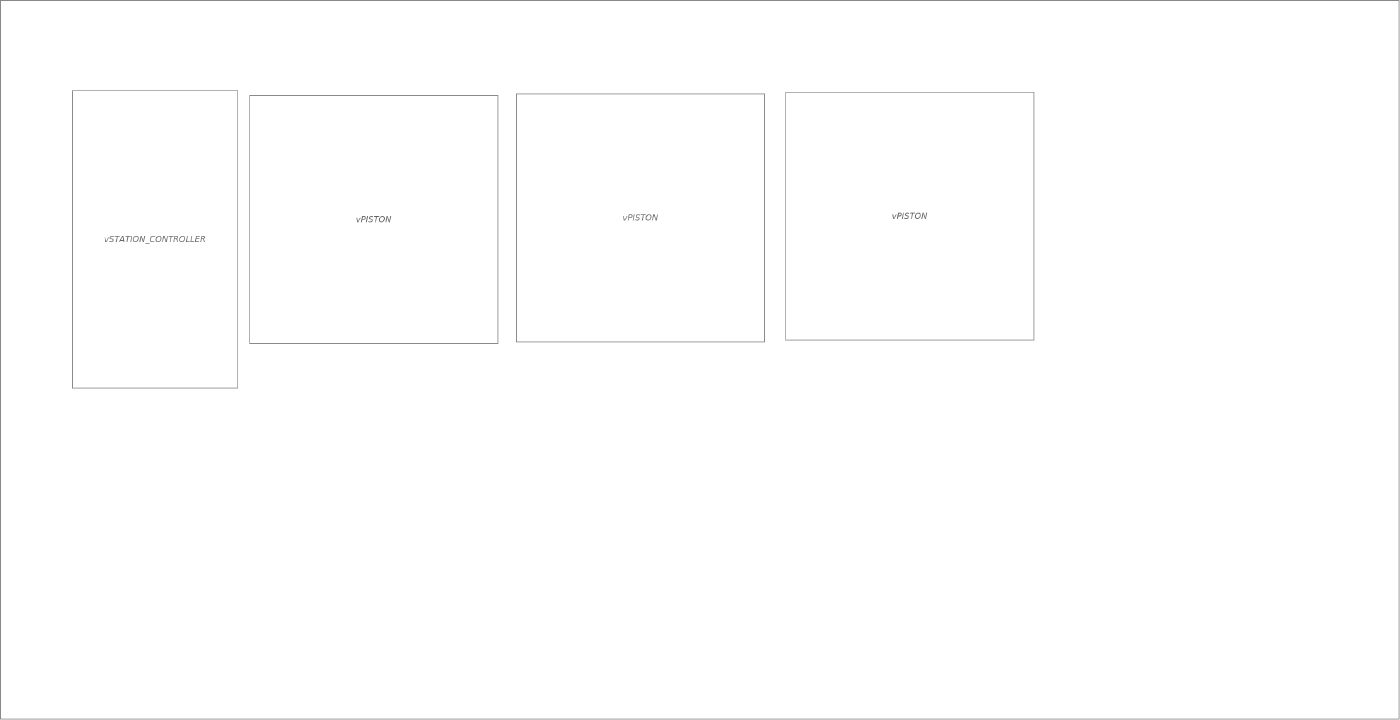
VISUALIZATION vSEPARATE  // 1690x870
VAR_IN_OUT
	vSEPARATE: FB_SEPARATE;
END_VAR
    Frame (301,115 300x300)
        shows vPISTON(PIST1 := vFEEDER.fbPIST1)
    Frame (623,113 300x300)
        shows vPISTON(PIST1 := vFEEDER.fbPIST2)
    Frame (948,111 300x300)
        shows vPISTON(PIST1 := vFEEDER.fbPIST3)
    Frame (87,109 200x360)
        shows vSTATION_CONTROLLER(vSTATION := vFEEDER)
END_VISUALIZATION

(* stored: Version 1.1.0.1, ProductVersion 3.1.4024.12
   Visu vSEPARATE: Id {629d8ca2-a747-40ec-bcb5-558372a8f264} *)
